(*Implements MoveRequest interface for EPICS Motor*)
FUNCTION_BLOCK FB_EpicsMoveRequest IMPLEMENTS I_MoveRequest
VAR
   // EPICS Interface
    {attribute 'no_copy'}
    stMotionCommand : REFERENCE TO ST_MotionCommand;
	{attribute 'no_copy'}
	stMotionStatus:  REFERENCE TO ST_MotionStatus;
	
    eEnableMode: E_StageEnableMode:=E_StageEnableMode.DURING_MOTION;
    {attribute 'hide'}
    eHomeMode	: E_EpicsHomeCmd := E_EpicsHomeCmd.NONE;
    {attribute 'hide'}
    bEnableDone : BOOL;
    {attribute 'hide'}
    bMoveOk: BOOL;
    (* non epics*)
    {attribute 'hide'}
    bExecute : BOOL;
    {attribute 'hide'}
    rtMoveCmdShortcut: R_TRIG;
    {attribute 'hide'}
    rtHomeCmdShortcut: R_TRIG;
    {attribute 'hide'}
    rtEnableMode: R_TRIG;
    {attribute 'hide'}
    rtNewMoveReq: R_TRIG;
    {attribute 'hide'}
    rtUserExec: R_TRIG;
    {attribute 'hide'}
    rtExec : R_TRIG;
    {attribute 'hide'}
    stMotionRequestStatus : ST_MoveRequestStatus;
    {attribute 'hide'}
    ftStopExec: F_TRIG;
    {attribute 'hide'}
    eRestoreSettingsState : ( RestoreSettingWaiting:=0, RestoreSettingDone:=1);
	rtExecute : R_TRIG;
END_VAR

// --- Validate command and status references ---
IF NOT __ISVALIDREF(stMotionCommand) OR NOT __ISVALIDREF(stMotionStatus) THEN
   RETURN;
END_IF

// --- Handle PLC shortcut commands (testing/circumvention logic) ---
rtMoveCmdShortcut(CLK := stMotionCommand.bMoveCmd);
rtHomeCmdShortcut(CLK := stMotionCommand.bHomeCmd);

// --- Rising edge of move command: issue MOVE_ABSOLUTE ---
IF rtMoveCmdShortcut.Q AND NOT bExecute THEN
    bExecute := TRUE;
    stMotionCommand.nCommand := E_EpicsMotorCmd.MOVE_ABSOLUTE;

// --- Rising edge of home command: validate and set HOME mode ---
ELSIF rtHomeCmdShortcut.Q AND NOT bExecute THEN
    IF IsValidHomeCmd(stMotionCommand.nCmdData) THEN
        IF stMotionCommand.nCmdData = E_EpicsHomeCmd.NONE THEN
            bExecute := FALSE; // Do not execute
        ELSE
            bExecute := TRUE;  // Valid home: enable
        END_IF
        stMotionCommand.nCommand := E_EpicsMotorCmd.HOME;
    END_IF
END_IF

// --- User/EPICS main exec entry ---
rtUserExec(CLK := bExecute);

// --- New move request: rising edge, axis not busy, no error, and interlocks OK ---
stMotionRequestStatus.bNewMoveReq S= NOT stMotionStatus.bBusy AND rtUserExec.Q AND NOT stMotionStatus.bError AND bMoveOk;

// --- New move stays active until execute ends or error occurs ---
stMotionRequestStatus.bNewMoveReq R= NOT bExecute OR stMotionStatus.bError;

// --- Prepare disable on end of move ---
stMotionRequestStatus.bPrepareDisable R= stMotionRequestStatus.bNewMoveReq;
rtNewMoveReq(CLK := stMotionRequestStatus.bNewMoveReq);

// --- Latch command data/type at queue entry, and check homing prerequisites ---
IF rtUserExec.Q THEN
    stMotionRequestStatus.nCmdData := stMotionCommand.nCmdData;
    stMotionRequestStatus.nCommand := stMotionCommand.nCommand;
    IF NOT stMotionCommand.bHomeCmd THEN
        IF eHomeMode <> E_EpicsHomeCmd.NONE AND NOT stMotionStatus.bHomed THEN
            stMotionStatus.sErrorMessage := 'Axis homing mode set, but homing routine pending';
        END_IF
    END_IF
END_IF

// --- Enable logic based on requested enable mode ---
rtEnableMode(CLK := (eEnableMode = E_StageEnableMode.DURING_MOTION));
CASE eEnableMode OF
    E_StageEnableMode.ALWAYS:
        stMotionRequestStatus.bEnable := NOT stMotionStatus.bError AND bMoveOk;
    E_StageEnableMode.DURING_MOTION:
        IF rtEnableMode.Q THEN
            stMotionRequestStatus.bEnable := FALSE; // DuringMotion disables enable on falling edge
        END_IF
        IF rtNewMoveReq.Q THEN
            stMotionRequestStatus.bEnable S= stMotionRequestStatus.bNewMoveReq;
        END_IF
END_CASE

// --- Execute if: not error, Execute set, and axis ready ---
stMotionRequestStatus.bExecute := NOT stMotionStatus.bError AND bExecute AND bEnableDone;
stMotionRequestStatus.bExecHome := stMotionRequestStatus.bExecute AND stMotionRequestStatus.nCommand = E_EpicsMotorCmd.HOME;
stMotionRequestStatus.bExecMove := stMotionRequestStatus.bExecute AND NOT stMotionRequestStatus.bExecHome;

// --- Latch axis busy at execute (clear done, busy, error) ---
rtExecute(CLK := bExecute);
IF rtExecute.Q THEN
    InitMoveRequest();
END_IF

// --- Clear local/EPICS interface --- 
stMotionCommand.bMoveCmd := FALSE;
stMotionCommand.bHomeCmd := FALSE;

// --- Prepare to disable at the end of execution (on falling edge) ---
ftStopExec(CLK := bExecute);
stMotionRequestStatus.bPrepareDisable S= (eEnableMode = E_StageEnableMode.DURING_MOTION) AND ftStopExec.Q;

// --- Reset error message on busy; optional: else show string on error condition ---
IF stMotionStatus.bBusy THEN
    stMotionStatus.sErrorMessage := '';
END_IF

METHOD PUBLIC CallAfterInit
VAR_INPUT
    stMotionCommand : REFERENCE TO ST_MotionCommand;
	stMotionStatus:  REFERENCE TO ST_MotionStatus;
END_VAR
THIS^.stMotionCommand REF=stMotionCommand;
THIS^.stMotionStatus REF=stMotionStatus;
END_METHOD

METHOD ClearMoveRequest
// falling edge here when target is reached, move halted
bExecute := FALSE;
stMotionStatus.bDone := FALSE;
stMotionStatus.bBusy := FALSE;
// release the cmds
stMotionCommand.bHomeCmd:=FALSE;
stMotionCommand.bMoveCmd:=FALSE;
END_METHOD

METHOD ClearMoveRequestErrors
stMotionStatus.bError := FALSE;
stMotionStatus.nErrorId := 0;
stMotionStatus.sErrorMessage := '';
stMotionRequestStatus.bExecute := FALSE;
END_METHOD

PROPERTY EnableMode : ENUM_StageEnableMode
GET
EnableMode := eEnableMode;
END_GET
SET
eEnableMode := EnableMode;
END_SET
END_PROPERTY

//FB_Init is always available implicitly and it is used primarily for initialization.
//The return value is not evaluated. For a specific influence, you can also declare the
//methods explicitly and provide additional code there with the standard initialization
//code. You can evaluate the return value.
METHOD FB_Init: BOOL
VAR_INPUT
    bInitRetains: BOOL; // TRUE: the retain variables are initialized (reset warm / reset cold)
    bInCopyCode: BOOL;  // TRUE: the instance will be copied to the copy code afterward (online change)
    stMotionCommand : REFERENCE TO ST_MotionCommand;
	stMotionStatus:  REFERENCE TO ST_MotionStatus;
END_VAR
THIS^.stMotionCommand REF=stMotionCommand;
THIS^.stMotionStatus REF=stMotionStatus;
END_METHOD

METHOD InitMoveRequest
stMotionStatus.bBusy := TRUE;
stMotionStatus.bDone := FALSE;
// reset error flag
stMotionStatus.sErrorMessage := '';
END_METHOD

METHOD IsValidHomeCmd : BOOL
VAR_INPUT
    CmdData : INT;
END_VAR
CASE CmdData OF
    E_EpicsHomeCmd.LOW_LIMIT,
    E_EpicsHomeCmd.HIGH_LIMIT,
    E_EpicsHomeCmd.HOME_VIA_LOW,
    E_EpicsHomeCmd.HOME_VIA_HIGH,
    E_EpicsHomeCmd.ABSOLUTE_SET,
    E_EpicsHomeCmd.AUTOZERO,
    E_EpicsHomeCmd.CURRENT_POSITION_METHOD,
    E_EpicsHomeCmd.NONE:
        IsValidHomeCmd := TRUE;
    ELSE
        IsValidHomeCmd := FALSE;
END_CASE
END_METHOD

METHOD MoveRequest
VAR_INPUT
    // From Axis through the drive
    EnableDone	: BOOL;
    // From Interlock through the drive
    MoveOk  : BOOL;
END_VAR
THIS^.bMoveOk := MoveOk;
THIS^.bEnableDone := EnableDone;
END_METHOD

(*Internal use only purpose*)
METHOD INTERNAL MoveRequestCmds
VAR_INPUT
    (* From Drive*)
    HomeCmd		: BOOL;
    MoveCmd		: BOOL;
	MoveOk 		: BOOL;
	EnableDone  : BOOL;
    HomeMode	: INT := E_EpicsHomeCmd.NONE;
    EnableMode	: E_StageEnableMode :=  E_StageEnableMode.DURING_MOTION;
END_VAR
THIS^.stMotionCommand.bHomeCmd := HomeCmd;
THIS^.stMotionCommand.nCmdData := HomeMode;
THIS^.stMotionCommand.bMoveCmd	:= MoveCmd;
THIS^.bMoveOk := MoveOk;
THIS^.bEnableDone := EnableDone;
THIS^.eEnableMode := EnableMode;
END_METHOD

METHOD MoveRequestCompleted
VAR_INPUT
    MoveDone : BOOL;
    HomeDone : BOOL;
END_VAR
stMotionStatus.bHomed := HomeDone;
ClearMoveRequest();
MoveRequestDone(Done:=MoveDone OR HomeDone);
END_METHOD

METHOD MoveRequestDone
VAR_INPUT
    Done : BOOL;
END_VAR
stMotionStatus.bDone := Done;
END_METHOD

METHOD MoveRequestError
VAR_INPUT
    Error :BOOL;
    ErrorId :UDINT;
    ErrorMessage:T_MAXSTRING;
END_VAR
stMotionStatus.bError := Error;
stMotionStatus.nErrorId := ErrorId;
stMotionStatus.sErrorMessage:= ErrorMessage;

IF Error THEN
	ClearMoveRequest();
END_IF
END_METHOD

METHOD ResetMoveEnable : BOOL
IF stMotionRequestStatus.bPrepareDisable THEN
    IF THIS^.eEnableMode=E_StageEnableMode.DURING_MOTION THEN
        THIS^.stMotionRequestStatus.bEnable := FALSE;
		ResetMoveEnable := TRUE;
	ELSE
		ResetMoveEnable := FALSE;
    END_IF
    THIS^.stMotionRequestStatus.bPrepareDisable := FALSE;
END_IF
END_METHOD

METHOD RestoreSettings
VAR_INPUT
    RestoreDone : BOOL;
    SavedPosition : LREAL;
END_VAR
// no needed in production since the actual position is already set on the axis
// and epics status will get that last position
// use this to restore anything thats not an axisref paramter.

CASE eRestoreSettingsState OF
    RestoreSettingWaiting:
        IF RestoreDone THEN
            THIS^.stMotionCommand.fPosition := SavedPosition;
            eRestoreSettingsState := RestoreSettingDone;
        END_IF
    RestoreSettingDone:;

END_CASE
END_METHOD

PROPERTY INTERNAL RestoreSettingsState : UINT
GET
//RestoreSettingsState := eRestoreSettingsState;
END_GET
END_PROPERTY

PROPERTY Status : REFERENCE TO ST_MoveRequestStatus
GET
Status REF= stMotionRequestStatus;
END_GET
END_PROPERTY

METHOD StopMoveRequest
THIS^.bExecute := FALSE;
END_METHOD

END_FUNCTION_BLOCK

(* stored: Version 1.1.0.1
   POU FB_EpicsMoveRequest: Id {f9713c0b-09a1-45a0-9fc6-342a7422cfa5}, SpecialFunc None
   Method CallAfterInit: Id {c5f4a41a-2a36-4ec0-b020-e8f39761af26}
   Method ClearMoveRequest: Id {fc3a5981-a4d7-4a2d-bb30-c09c583c9e55}
   Method ClearMoveRequestErrors: Id {2bb41509-e70c-4465-a06c-a29812268b06}
   Property EnableMode: Id {9356bd40-5ede-4c8b-b065-3ca414d58ac7}
   Get Get: Id {0f06a9c5-786f-4b36-9ffb-1932b02bcacd}
   Set Set: Id {21b092e9-96af-46ee-9d8d-c77dcd117d11}
   Method FB_Init: Id {9133e91c-1e17-4b3b-aa68-c9be539e6510}
   Method InitMoveRequest: Id {2d590fc6-f95b-45d5-9e1d-141474a0f09b}
   Method IsValidHomeCmd: Id {ee32dcd3-ada0-4e13-b5c7-6e8287ec8a3c}
   Method MoveRequest: Id {664b6655-0949-47c1-b45f-a64c7d0cda3b}
   Method MoveRequestCmds: Id {d84ff316-c87c-445b-b337-4ae6bc661e04}
   Method MoveRequestCompleted: Id {29932e68-9af9-4521-bd55-b747e571b46c}
   Method MoveRequestDone: Id {ab10537f-2bb4-4a28-9c3a-e3028ea8d9fc}
   Method MoveRequestError: Id {674719eb-75b4-4cc3-924b-ecc3d1af31ff}
   Method ResetMoveEnable: Id {f28760d0-5752-4bf4-b850-362b1de6a659}
   Method RestoreSettings: Id {08281416-55cb-4b9c-81b3-3cf6fd0d7faf}
   Property RestoreSettingsState: Id {b366cb5d-502b-43b3-8623-320516670b00}
   Get Get: Id {a39741db-d8b0-422d-b3ab-4a4dba01333b}
   Property Status: Id {f678d159-cc5d-41ad-889c-5f951c755b6f}
   Get Get: Id {08876ea6-b526-4166-bd4c-0a2aa1b11215}
   Method StopMoveRequest: Id {92e9d903-c05e-4a96-bba3-dd1393b47659} *)
